{attribute 'qualified_only'}
VAR_GLOBAL PERSISTENT
	aComboboxRecipes : ARRAY [1..100] OF stComboBoxRecipes;
	RecetaEditar:RecetaEdicion;
	EdicionRecetaNro:INT;
	GrabarRecetaEdicion:BOOL;
	LeerRecetaEditar:BOOL;
	BibliotecaRecetas:ARRAY [1..100] OF RecetaEdicion;
END_VAR

(* stored: Version 1.1.0.1, ProductVersion 3.1.4024.13
   GVL RecetasGestion: Id {0a3a7191-7561-4e84-b227-6c96e73f52a4} *)
